// Mitsubishi GX Works2 project: group3_tes2t   PLC: FX3G

// global labels: Global1
VAR_GLOBAL
  morning_switch AT X007 : BOOL;
  break_switch AT X005 : BOOL;
  materials_stock AT M1 : BOOL;
  morning_light AT Y007 : BOOL;
END_VAR
VAR_GLOBAL CONSTANT
  reset_analog_output : INT;
END_VAR
VAR_GLOBAL
  analog_output_reset AT D8282 : INT;
END_VAR
VAR_GLOBAL CONSTANT
  reset_analog_input : INT;
  reset_constant0 : INT;
END_VAR
VAR_GLOBAL
  day_switch AT X007 : BOOL;
  day_light AT Y007 : BOOL;
  analog_output AT D8282 : INT;
  check_material AT M2 : BOOL;
  petel_input AT D1100 : REAL;
END_VAR
VAR_GLOBAL CONSTANT
  min_petel : REAL := 280.0;
END_VAR
VAR_GLOBAL
  lemon_input AT D1200 : REAL;
END_VAR
VAR_GLOBAL CONSTANT
  min_lemon : REAL := 455.0;
END_VAR
VAR_GLOBAL
  gummy_input AT D1300 : REAL;
  stabilizer_input AT D1400 : REAL;
  dgima_kind AT X001 : BOOL;
END_VAR
VAR_GLOBAL CONSTANT
  lemol_7_pinuk : REAL;
  lemon_7_pinuk : REAL := 665;
  gummy_7_pinuk : REAL := 70;
  petel_7_pinuk : REAL := 385;
  stabilizer_7_pinuk : REAL := 210;
END_VAR
VAR_GLOBAL
  check_pinuk AT M3 : BOOL;
  analog_input AT D8280 : INT;
END_VAR
VAR_GLOBAL CONSTANT
  normalizer : REAL := 400;
END_VAR
VAR_GLOBAL
  glida_type AT D1500 : REAL;
END_VAR
VAR_GLOBAL CONSTANT
  min_ragil : REAL;
  min_pinuk : REAL := 6.0;
  max_ragil : REAL := 5.0;
  max_pinuk : REAL := 10.0;
END_VAR
VAR_GLOBAL
  ragil_choose AT M4 : BOOL;
  pinuk_choose AT M5 : BOOL;
  cooking_timer AT TC1 : BOOL;
END_VAR
VAR_GLOBAL CONSTANT
  cooking_duration : INT := 50;
END_VAR
VAR_GLOBAL
  end_cooking AT TS1 : BOOL;
  cooking_light AT Y000 : BOOL;
  making_light AT Y000 : BOOL;
  end_making AT TS1 : BOOL;
  making_timer AT TC1 : BOOL;
END_VAR
VAR_GLOBAL CONSTANT
  making_duration : INT := 50;
  petel_ragil_ice_weight : REAL := 350;
END_VAR
VAR_GLOBAL
  petel_making_con AT D1600 : REAL;
END_VAR
VAR_GLOBAL CONSTANT
  lemon_ragil_ice_weight : REAL := 490;
END_VAR
VAR_GLOBAL
  lemon_making_con AT D1610 : REAL;
END_VAR
VAR_GLOBAL CONSTANT
  petel_pinuk_ice_weight : REAL := 560;
  lemon_pinuk_ice_weight : REAL := 700;
END_VAR
VAR_GLOBAL
  petel_stock AT D1110 : REAL;
  lemon_stock AT D1210 : REAL;
  gummy_stock AT D1310 : REAL;
  stabilizer_stock AT D1410 : REAL;
END_VAR
VAR_GLOBAL CONSTANT
  min_stabilizer1 : REAL := 105;
  min_gummy1 : REAL := 28.0;
END_VAR
VAR_GLOBAL
  petel_freeze_con AT D1700 : REAL;
  lemon_freeze_con AT D1710 : REAL;
  start_freeze AT X002 : BOOL;
  test_light AT M25 : BOOL;
  freezing_timer AT TC2 : BOOL;
END_VAR
VAR_GLOBAL CONSTANT
  freezing_duration : INT := 80;
END_VAR
VAR_GLOBAL
  end_freezing AT TS2 : BOOL;
  freezing_light AT Y002 : BOOL;
  temp_sensor AT X003 : BOOL;
  mix_con AT D1800 : REAL;
  mixRagil AT TC3 : BOOL;
END_VAR
VAR_GLOBAL CONSTANT
  timeRagil : INT := 30;
END_VAR
VAR_GLOBAL
  mixPinuk AT TC4 : BOOL;
END_VAR
VAR_GLOBAL CONSTANT
  timePinuk : INT := 50;
END_VAR
VAR_GLOBAL
  finish_mix_ragil AT TS3 : BOOL;
  finish_mix_pinuk AT TS4 : BOOL;
  helper AT M0 : BOOL;
  first_lamp AT TS5 : BOOL;
  first AT Y005 : BOOL;
  second_lamp AT TS6 : BOOL;
  second AT Y006 : BOOL;
  on_of_mix AT TC6 : BOOL;
  on_of_mix2 AT TC6 : BOOL;
END_VAR
VAR_GLOBAL CONSTANT
  on_off : INT := 5;
END_VAR
VAR_GLOBAL
  on_off_mix2 AT TC6 : BOOL;
  on_off_mix AT TC5 : BOOL;
  start_packing AT X004 : BOOL;
  packCone AT X000 : BOOL;
  first_packed AT CS0 : BOOL;
  seventh_packed AT CS1 : BOOL;
  pack_6_more AT Y004 : BOOL;
  count_first_cone AT CC0 : BOOL;
END_VAR
VAR_GLOBAL CONSTANT
  counter_first : INT := 1;
  first_counter : REAL := 1;
END_VAR
VAR_GLOBAL
  count_6_cones AT CC1 : BOOL;
  count_6_more AT CC1 : BOOL;
END_VAR
VAR_GLOBAL CONSTANT
  counter_six : INT := 7;
END_VAR
VAR_GLOBAL
  end_one_iteration AT M6 : BOOL;
  inventory AT D1900 : REAL;
END_VAR
VAR_GLOBAL CONSTANT
  add_one_packed : REAL := 1;
END_VAR
VAR_GLOBAL
  day_end AT M7 : BOOL;
  check_ragil AT M2 : BOOL;
  end_of_stock AT M8 : BOOL;
  inventory_4_output AT D2000 : REAL;
  start_mixing AT Y011 : BOOL;
  exception_day_end AT M9 : BOOL;
  gummy_added AT M10 : BOOL;
END_VAR
VAR_GLOBAL CONSTANT
  const_10 : REAL := 10.0;
  const_40 : REAL := 40;
END_VAR

// task Task_01 (event TRUE, interval 0, priority 31): POU_01

PROGRAM POU_01
(* structured ladder/FBD written out as ST: instructions are called as NAME(EN, inputs, outputs); _pN, _eN, _tN stand for wires *)
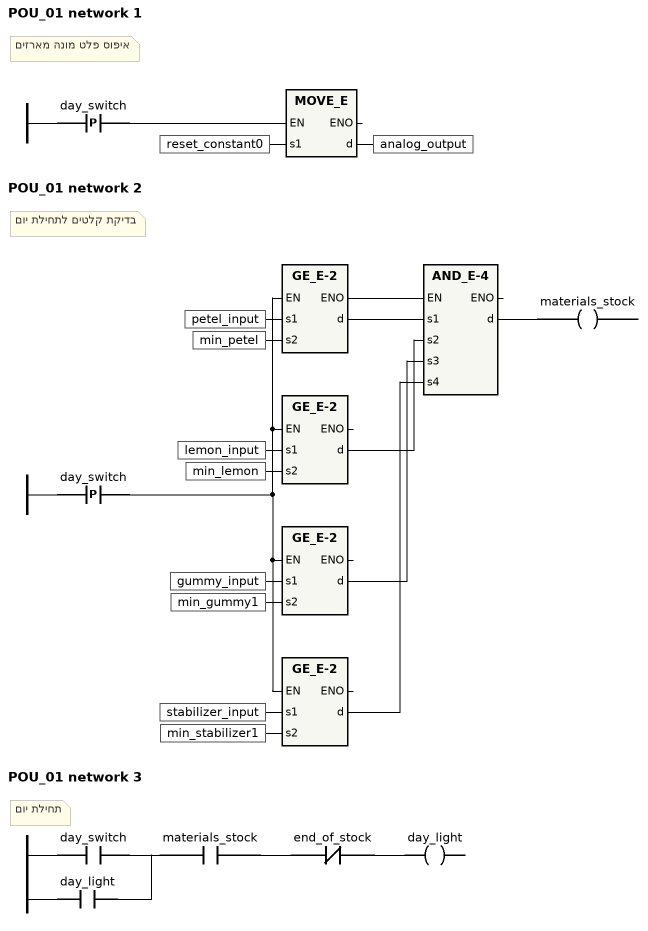
(* network 1 *)
(* איפוס פלט מונה מארזים *)
MOVE_E(LDP(TRUE, day_switch), reset_constant0, analog_output);
(* network 2 *)
(* בדיקת קלטים לתחילת יום *)
_p1 := LDP(TRUE, day_switch);
_e3 := GE_E(_p1, petel_input, min_petel, _t2);
GE_E(_p1, lemon_input, min_lemon, _t4);
GE_E(_p1, gummy_input, min_gummy1, _t5);
GE_E(_p1, stabilizer_input, min_stabilizer1, _t6);
AND_E(_e3, _t2, _t4, _t5, _t6, _t7);
materials_stock := _t7;
(* network 3 *)
(* תחילת יום *)
day_light := ((day_switch OR day_light) AND materials_stock) AND NOT end_of_stock;
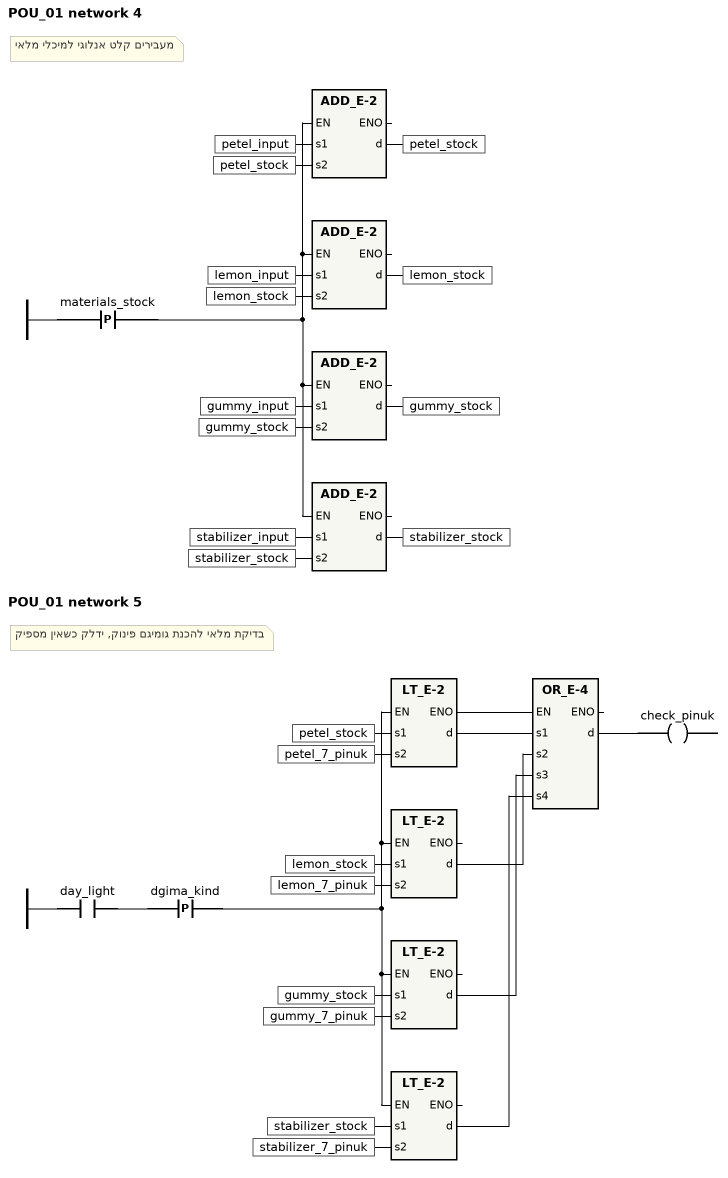
(* network 4 *)
(* מעבירים קלט אנלוגי למיכלי מלאי *)
_p1 := LDP(TRUE, materials_stock);
ADD_E(_p1, petel_input, petel_stock, petel_stock);
ADD_E(_p1, lemon_input, lemon_stock, lemon_stock);
ADD_E(_p1, gummy_input, gummy_stock, gummy_stock);
ADD_E(_p1, stabilizer_input, stabilizer_stock, stabilizer_stock);
(* network 5 *)
(* בדיקת מלאי להכנת גומיגם פינוק, ידלק כשאין מספיק *)
_p1 := day_light AND LDP(TRUE, dgima_kind);
_e3 := LT_E(_p1, petel_stock, petel_7_pinuk, _t2);
LT_E(_p1, lemon_stock, lemon_7_pinuk, _t4);
LT_E(_p1, gummy_stock, gummy_7_pinuk, _t5);
LT_E(_p1, stabilizer_stock, stabilizer_7_pinuk, _t6);
OR_E(_e3, _t2, _t4, _t5, _t6, _t7);
check_pinuk := _t7;
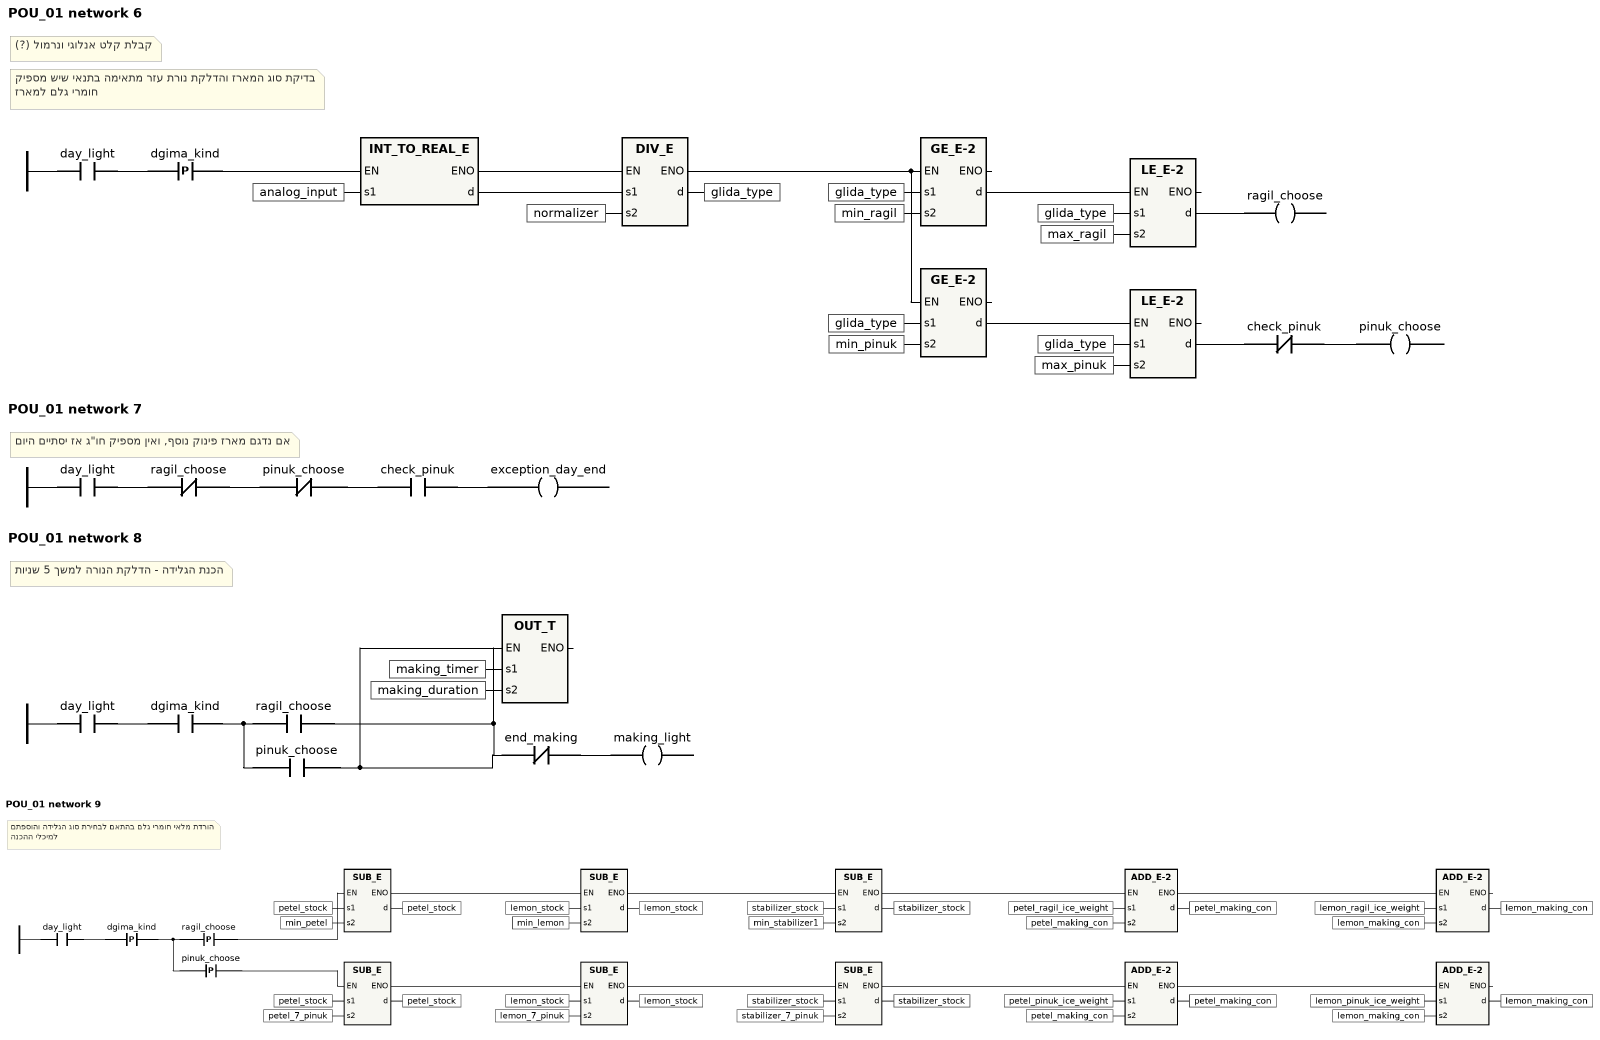
(* network 6 *)
(* קבלת קלט אנלוגי ונרמול (?) *)
(* בדיקת סוג המארז והדלקת נורת עזר מתאימה בתנאי שיש מספיק חומרי גלם למארז *)
_e2 := INT_TO_REAL_E(day_light AND LDP(TRUE, dgima_kind), analog_input, _t1);
_e3 := DIV_E(_e2, _t1, normalizer, glida_type);
GE_E(_e3, glida_type, min_ragil, _t4);
LE_E(_t4, glida_type, max_ragil, _t5);
ragil_choose := _t5;
GE_E(_e3, glida_type, min_pinuk, _t6);
LE_E(_t6, glida_type, max_pinuk, _t7);
pinuk_choose := _t7 AND NOT check_pinuk;
(* network 7 *)
(* אם נדגם מארז פינוק נוסף, ואין מספיק חו"ג אז יסתיים היום *)
exception_day_end := day_light AND NOT ragil_choose AND NOT pinuk_choose AND check_pinuk;
(* network 8 *)
(* הכנת הגלידה - הדלקת הנורה למשך 5 שניות *)
_p1 := day_light AND dgima_kind;
_p2 := (_p1 AND ragil_choose) OR (_p1 AND pinuk_choose);
OUT_T(_p2, making_timer, making_duration);
making_light := _p2 AND NOT end_making;
(* network 9 *)
(* הורדת מלאי חומרי גלם בהתאם לבחירת סוג הגלידה והוספתם למיכלי ההכנה *)
_p1 := day_light AND LDP(TRUE, dgima_kind);
_e2 := SUB_E(_p1 AND LDP(TRUE, ragil_choose), petel_stock, min_petel, petel_stock);
_e3 := SUB_E(_e2, lemon_stock, min_lemon, lemon_stock);
_e4 := SUB_E(_e3, stabilizer_stock, min_stabilizer1, stabilizer_stock);
_e5 := ADD_E(_e4, petel_ragil_ice_weight, petel_making_con, petel_making_con);
ADD_E(_e5, lemon_ragil_ice_weight, lemon_making_con, lemon_making_con);
_e6 := SUB_E(_p1 AND LDP(TRUE, pinuk_choose), petel_stock, petel_7_pinuk, petel_stock);
_e7 := SUB_E(_e6, lemon_stock, lemon_7_pinuk, lemon_stock);
_e8 := SUB_E(_e7, stabilizer_stock, stabilizer_7_pinuk, stabilizer_stock);
_e9 := ADD_E(_e8, petel_pinuk_ice_weight, petel_making_con, petel_making_con);
ADD_E(_e9, lemon_pinuk_ice_weight, lemon_making_con, lemon_making_con);
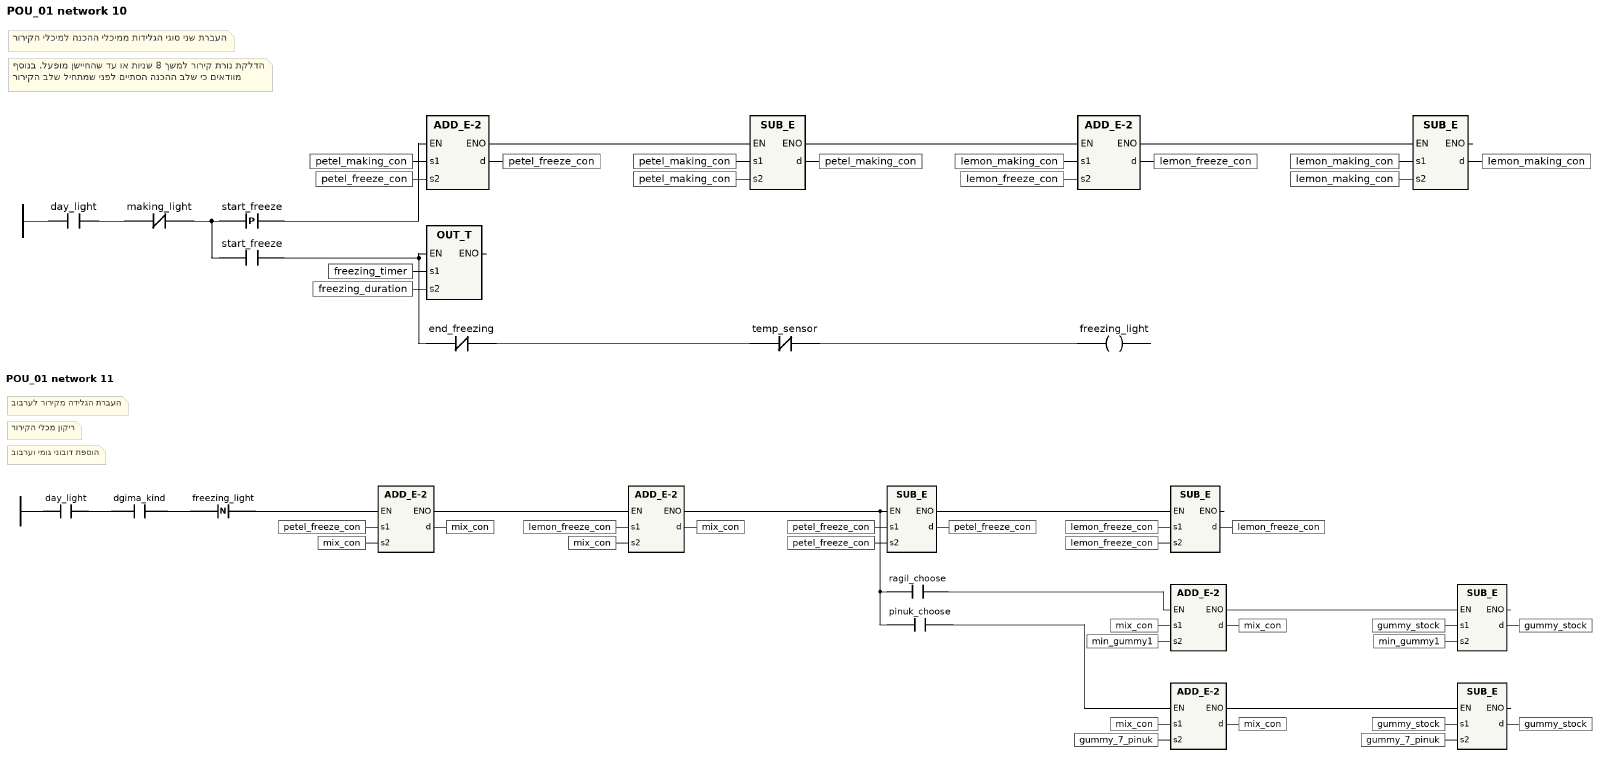
(* network 10 *)
(* העברת שני סוגי הגלידות ממיכלי ההכנה למיכלי הקירור *)
(* הדלקת נורת קירור למשך 8 שניות או עד שהחיישן מופעל. בנוסף מוודאים כי שלב ההכנה הסתיים לפני שמתחיל שלב הקירור *)
_p1 := day_light AND NOT making_light;
_e2 := ADD_E(_p1 AND LDP(TRUE, start_freeze), petel_making_con, petel_freeze_con, petel_freeze_con);
_e3 := SUB_E(_e2, petel_making_con, petel_making_con, petel_making_con);
_e4 := ADD_E(_e3, lemon_making_con, lemon_freeze_con, lemon_freeze_con);
SUB_E(_e4, lemon_making_con, lemon_making_con, lemon_making_con);
_p5 := _p1 AND start_freeze;
OUT_T(_p5, freezing_timer, freezing_duration);
freezing_light := _p5 AND NOT end_freezing AND NOT temp_sensor;
(* network 11 *)
(* העברת הגלידה מקירור לערבוב *)
(* ריקון מכלי הקירור *)
(* הוספת דובוני גומי וערבוב *)
_e1 := ADD_E(day_light AND dgima_kind AND LDF(TRUE, freezing_light), petel_freeze_con, mix_con, mix_con);
_e2 := ADD_E(_e1, lemon_freeze_con, mix_con, mix_con);
_e3 := SUB_E(_e2, petel_freeze_con, petel_freeze_con, petel_freeze_con);
SUB_E(_e3, lemon_freeze_con, lemon_freeze_con, lemon_freeze_con);
_e4 := ADD_E(_e2 AND ragil_choose, mix_con, min_gummy1, mix_con);
SUB_E(_e4, gummy_stock, min_gummy1, gummy_stock);
_e5 := ADD_E(_e2 AND pinuk_choose, mix_con, gummy_7_pinuk, mix_con);
SUB_E(_e5, gummy_stock, gummy_7_pinuk, gummy_stock);
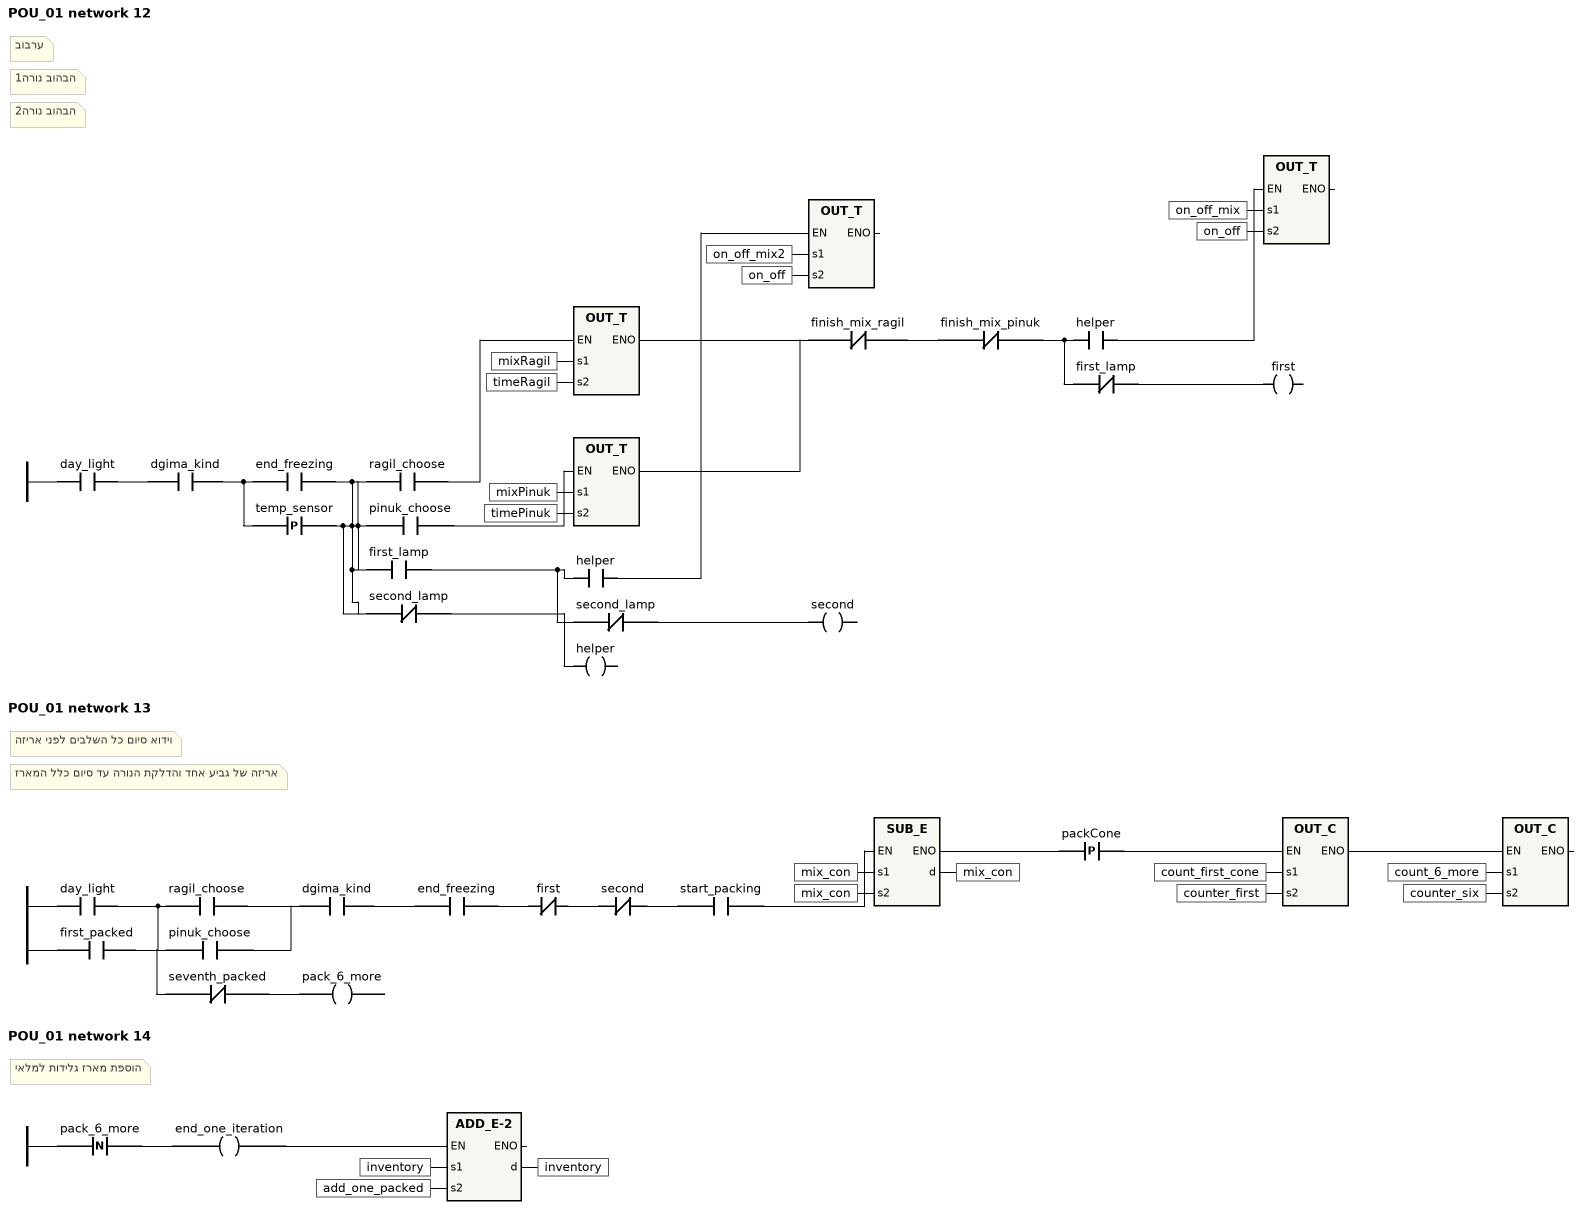
(* network 12 *)
(* ערבוב *)
(* הבהוב נורה1 *)
(* הבהוב נורה2 *)
_p1 := day_light AND dgima_kind;
_p2 := (_p1 AND end_freezing) OR (_p1 AND LDP(TRUE, temp_sensor));
_e3 := OUT_T(_p2 AND ragil_choose, mixRagil, timeRagil);
_e4 := OUT_T(_p2 AND pinuk_choose, mixPinuk, timePinuk);
_p5 := ((_e3 OR _e4) AND NOT finish_mix_ragil) AND NOT finish_mix_pinuk;
OUT_T(_p5 AND helper, on_off_mix, on_off);
first := _p5 AND NOT first_lamp;
_p6 := _p2 AND first_lamp;
OUT_T(_p6 AND helper, on_off_mix2, on_off);
second := _p6 AND NOT second_lamp;
helper := _p2 AND NOT second_lamp;
(* network 13 *)
(* וידוא סיום כל השלבים לפני אריזה *)
(* אריזה של גביע אחד והדלקת הנורה עד סיום כלל המארז *)
_e1 := SUB_E(((((((day_light AND ragil_choose) OR (day_light AND pinuk_choose)) AND dgima_kind) AND end_freezing) AND NOT first) AND NOT second) AND start_packing, mix_con, mix_con, mix_con);
_e2 := OUT_C(_e1 AND LDP(TRUE, packCone), count_first_cone, counter_first);
OUT_C(_e2, count_6_more, counter_six);
pack_6_more := first_packed AND NOT seventh_packed;
(* network 14 *)
(* הוספת מארז גלידות למלאי *)
_p1 := LDF(TRUE, pack_6_more);
end_one_iteration := _p1;
ADD_E(_p1, inventory, add_one_packed, inventory);
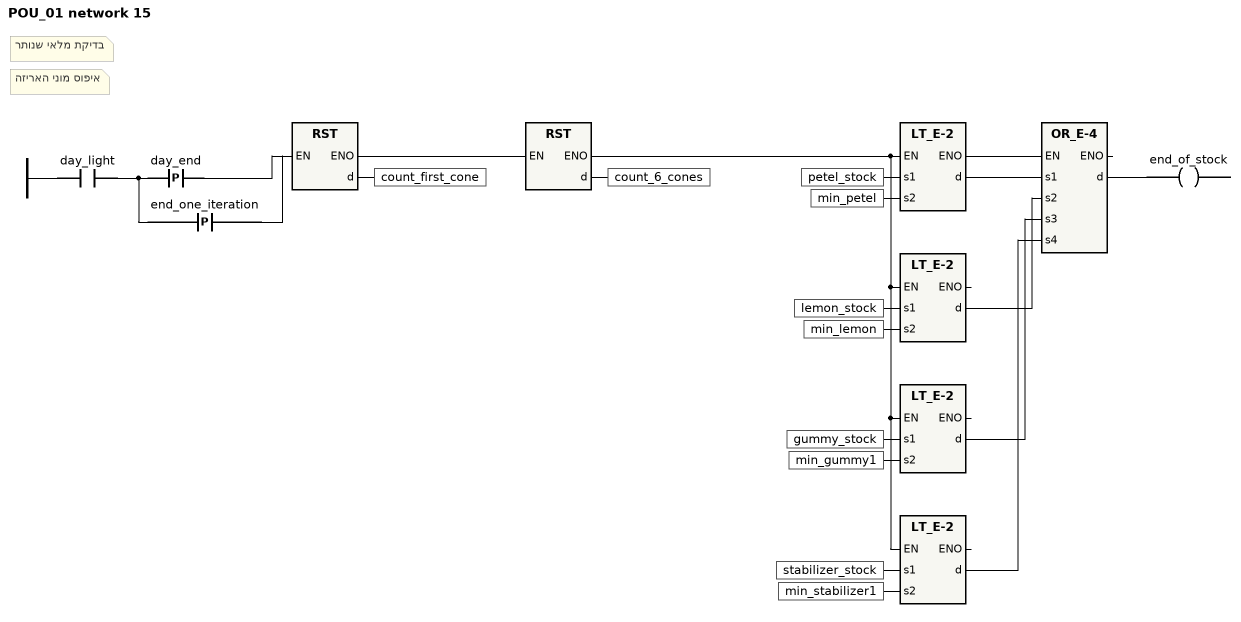
(* network 15 *)
(* בדיקת מלאי שנותר *)
(* איפוס מוני האריזה *)
_e1 := RST((day_light AND LDP(TRUE, day_end)) OR (day_light AND LDP(TRUE, end_one_iteration)), count_first_cone);
_e2 := RST(_e1, count_6_cones);
_e4 := LT_E(_e2, petel_stock, min_petel, _t3);
LT_E(_e2, lemon_stock, min_lemon, _t5);
LT_E(_e2, gummy_stock, min_gummy1, _t6);
LT_E(_e2, stabilizer_stock, min_stabilizer1, _t7);
OR_E(_e4, _t3, _t5, _t6, _t7, _t8);
end_of_stock := _t8;
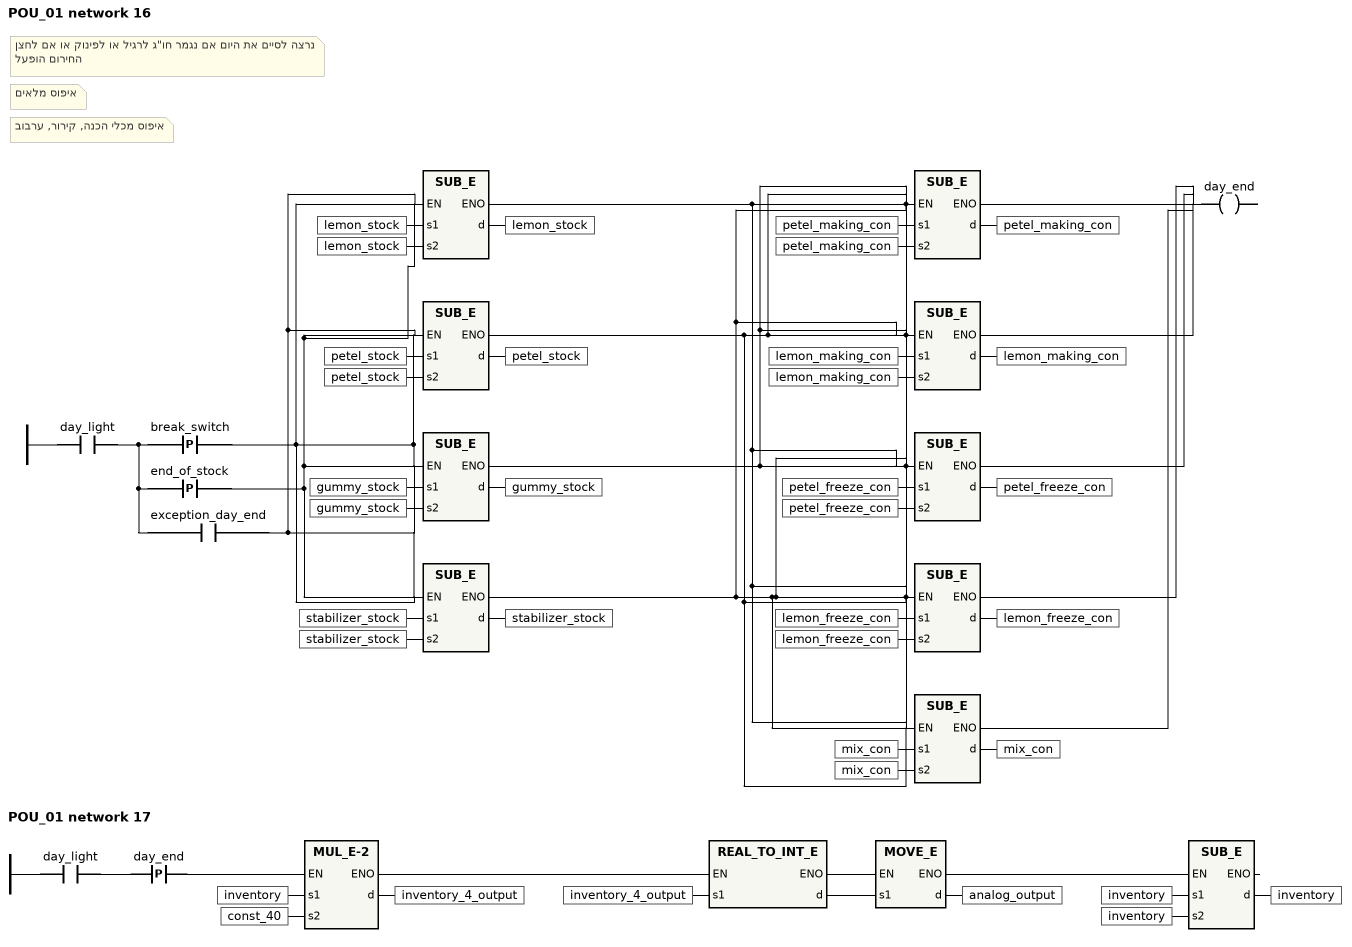
(* network 16 *)
(* נרצה לסיים את היום אם נגמר חו"ג לרגיל או לפינוק או אם לחצן החירום הופעל *)
(* איפוס מלאים *)
(* איפוס מכלי הכנה, קירור, ערבוב *)
_p1 := (day_light AND LDP(TRUE, break_switch)) OR (day_light AND LDP(TRUE, end_of_stock)) OR (day_light AND exception_day_end);
_e2 := SUB_E(_p1, lemon_stock, lemon_stock, lemon_stock);
_e3 := SUB_E(_p1, petel_stock, petel_stock, petel_stock);
_e4 := SUB_E(_p1, gummy_stock, gummy_stock, gummy_stock);
_e5 := SUB_E(_p1, stabilizer_stock, stabilizer_stock, stabilizer_stock);
_p6 := _e2 OR _e3 OR _e4 OR _e5;
_e7 := SUB_E(_p6, petel_making_con, petel_making_con, petel_making_con);
_e8 := SUB_E(_p6, lemon_making_con, lemon_making_con, lemon_making_con);
_e9 := SUB_E(_p6, petel_freeze_con, petel_freeze_con, petel_freeze_con);
_e10 := SUB_E(_p6, lemon_freeze_con, lemon_freeze_con, lemon_freeze_con);
_e11 := SUB_E(_p6, mix_con, mix_con, mix_con);
day_end := _e7 OR _e8 OR _e9 OR _e10 OR _e11;
(* network 17 *)
_e1 := MUL_E(day_light AND LDP(TRUE, day_end), inventory, const_40, inventory_4_output);
_e3 := REAL_TO_INT_E(_e1, inventory_4_output, _t2);
_e4 := MOVE_E(_e3, _t2, analog_output);
SUB_E(_e4, inventory, inventory, inventory);
END_PROGRAM
